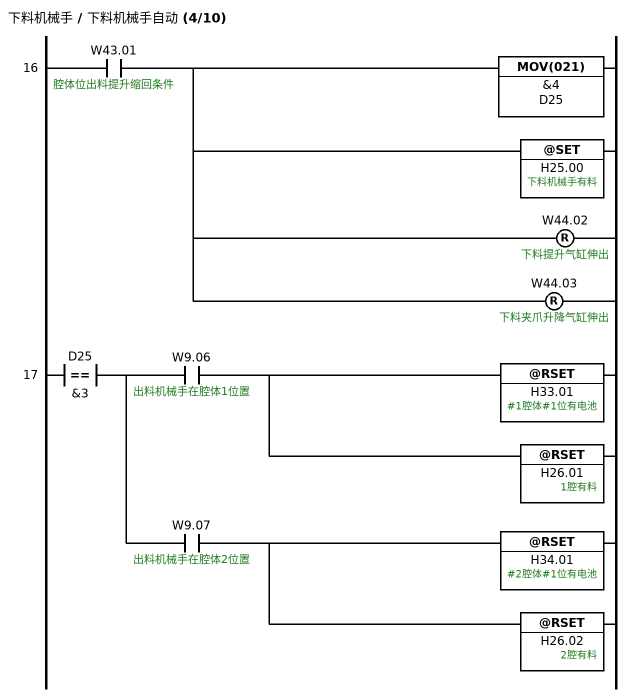
; [picture p168: 下料机械手 / 下料机械手自动, rungs 16-17]
; rung 16
LD W43.01  ; 腔体位出料提升缩回条件
MOV(021) &4 D25
@SET H25.00  ; 下料机械手有料
RSET W44.02  ; 下料提升气缸伸出
RSET W44.03  ; 下料夹爪升降气缸伸出
; rung 17
LD=(300) D25 &3
OUT TR0
AND W9.06  ; 出料机械手在腔体1位置
@RSET H33.01  ; #1腔体#1位有电池
@RSET H26.01  ; 1腔有料
LD TR0
AND W9.07  ; 出料机械手在腔体2位置
@RSET H34.01  ; #2腔体#1位有电池
@RSET H26.02  ; 2腔有料

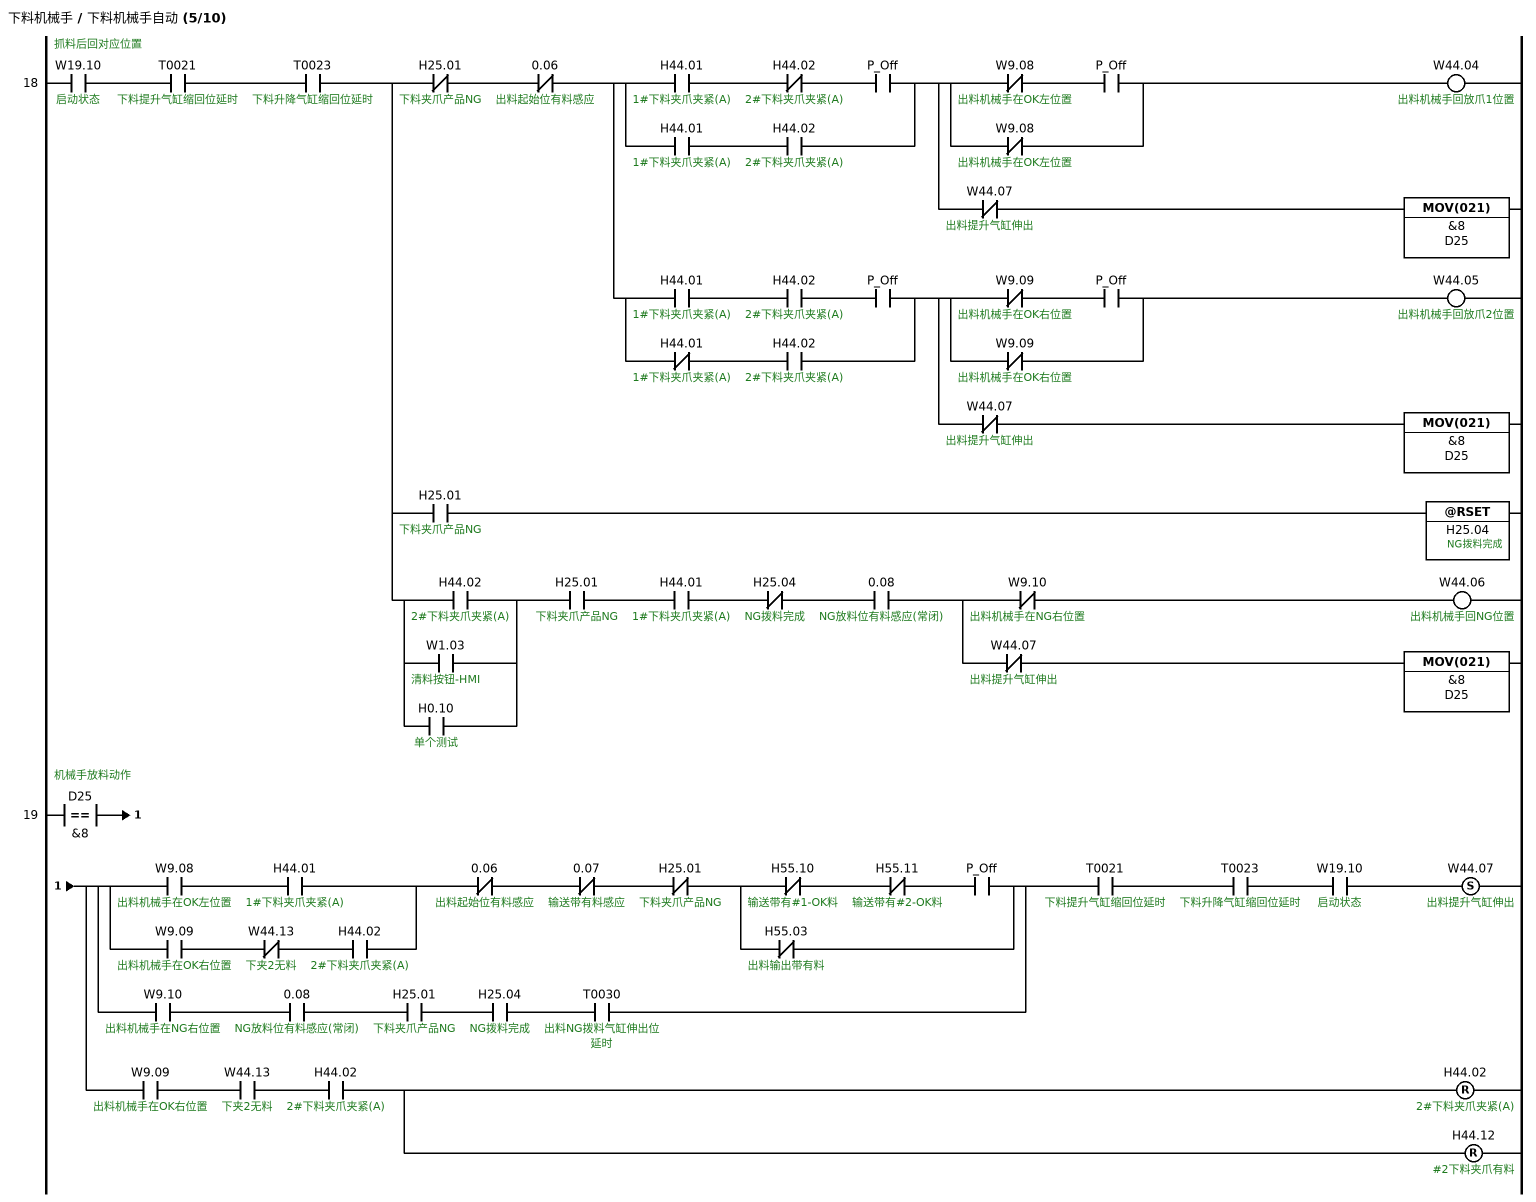
; rung 18: 抓料后回对应位置
LD W19.10  ; 启动状态
AND T0021  ; 下料提升气缸缩回位延时
AND T0023  ; 下料升降气缸缩回位延时
OUT TR0
ANDNOT H25.01  ; 下料夹爪产品NG
ANDNOT 0.06  ; 出料起始位有料感应
OUT TR1
LD H44.01  ; 1#下料夹爪夹紧(A)
ANDNOT H44.02  ; 2#下料夹爪夹紧(A)
AND P_Off
LD H44.01  ; 1#下料夹爪夹紧(A)
AND H44.02  ; 2#下料夹爪夹紧(A)
ORLD
ANDLD
OUT TR2
LDNOT W9.08  ; 出料机械手在OK左位置
AND P_Off
ORNOT W9.08  ; 出料机械手在OK左位置
ANDLD
OUT W44.04  ; 出料机械手回放爪1位置
LD TR2
ANDNOT W44.07  ; 出料提升气缸伸出
MOV(021) &8 D25
LD TR1
LD H44.01  ; 1#下料夹爪夹紧(A)
AND H44.02  ; 2#下料夹爪夹紧(A)
AND P_Off
LDNOT H44.01  ; 1#下料夹爪夹紧(A)
AND H44.02  ; 2#下料夹爪夹紧(A)
ORLD
ANDLD
OUT TR1
LDNOT W9.09  ; 出料机械手在OK右位置
AND P_Off
ORNOT W9.09  ; 出料机械手在OK右位置
ANDLD
OUT W44.05  ; 出料机械手回放爪2位置
LD TR1
ANDNOT W44.07  ; 出料提升气缸伸出
MOV(021) &8 D25
LD TR0
AND H25.01  ; 下料夹爪产品NG
@RSET H25.04  ; NG拨料完成
LD TR0
LD H44.02  ; 2#下料夹爪夹紧(A)
OR W1.03  ; 清料按钮-HMI
OR H0.10  ; 单个测试
ANDLD
AND H25.01  ; 下料夹爪产品NG
AND H44.01  ; 1#下料夹爪夹紧(A)
ANDNOT H25.04  ; NG拨料完成
AND 0.08  ; NG放料位有料感应(常闭)
OUT TR0
ANDNOT W9.10  ; 出料机械手在NG右位置
OUT W44.06  ; 出料机械手回NG位置
LD TR0
ANDNOT W44.07  ; 出料提升气缸伸出
MOV(021) &8 D25
; rung 19: 机械手放料动作
LD=(300) D25 &8
OUT TR0
LD W9.08  ; 出料机械手在OK左位置
AND H44.01  ; 1#下料夹爪夹紧(A)
LD W9.09  ; 出料机械手在OK右位置
ANDNOT W44.13  ; 下夹2无料
AND H44.02  ; 2#下料夹爪夹紧(A)
ORLD
ANDNOT 0.06  ; 出料起始位有料感应
ANDNOT 0.07  ; 输送带有料感应
ANDNOT H25.01  ; 下料夹爪产品NG
LDNOT H55.10  ; 输送带有#1-OK料
ANDNOT H55.11  ; 输送带有#2-OK料
AND P_Off
ORNOT H55.03  ; 出料输出带有料
ANDLD
LD W9.10  ; 出料机械手在NG右位置
AND 0.08  ; NG放料位有料感应(常闭)
AND H25.01  ; 下料夹爪产品NG
AND H25.04  ; NG拨料完成
AND T0030  ; 出料NG拨料气缸伸出位延时
ORLD
ANDLD
AND T0021  ; 下料提升气缸缩回位延时
AND T0023  ; 下料升降气缸缩回位延时
AND W19.10  ; 启动状态
SET W44.07  ; 出料提升气缸伸出
LD TR0
AND W9.09  ; 出料机械手在OK右位置
AND W44.13  ; 下夹2无料
AND H44.02  ; 2#下料夹爪夹紧(A)
RSET H44.02  ; 2#下料夹爪夹紧(A)
RSET H44.12  ; #2下料夹爪有料

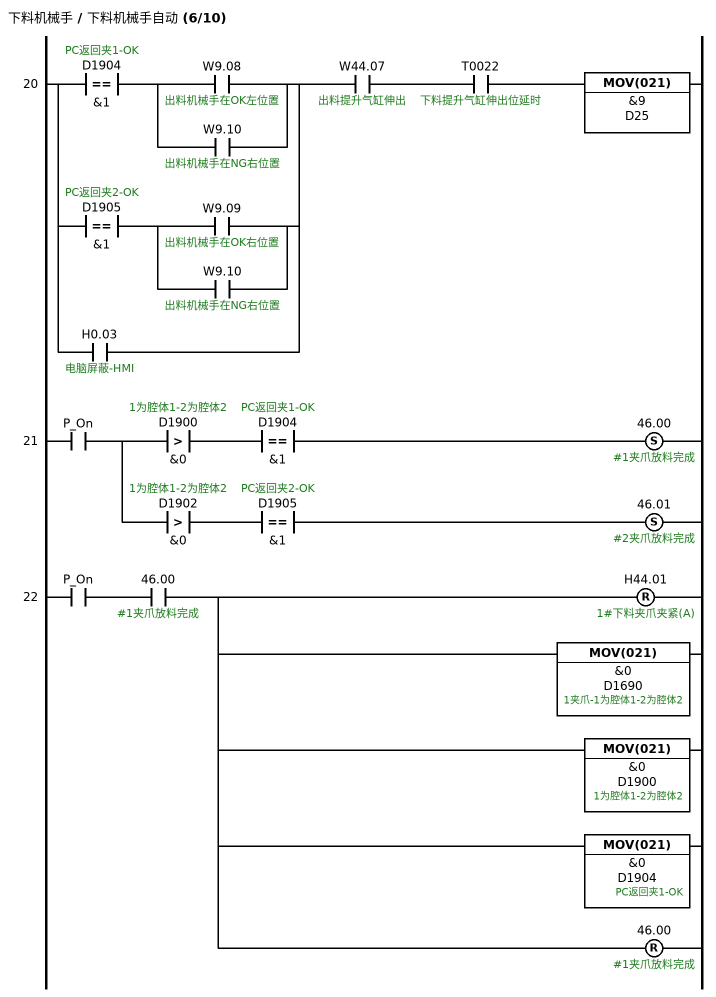
; rung 20
LD=(300) D1904 &1  ; PC返回夹1-OK
LD W9.08  ; 出料机械手在OK左位置
OR W9.10  ; 出料机械手在NG右位置
ANDLD
LD=(300) D1905 &1  ; PC返回夹2-OK
LD W9.09  ; 出料机械手在OK右位置
OR W9.10  ; 出料机械手在NG右位置
ANDLD
ORLD
OR H0.03  ; 电脑屏蔽-HMI
AND W44.07  ; 出料提升气缸伸出
AND T0022  ; 下料提升气缸伸出位延时
MOV(021) &9 D25
; rung 21
LD P_On
OUT TR0
AND>(320) D1900 &0  ; 1为腔体1-2为腔体2
AND=(300) D1904 &1  ; PC返回夹1-OK
SET 46.00  ; #1夹爪放料完成
LD TR0
AND>(320) D1902 &0  ; 1为腔体1-2为腔体2
AND=(300) D1905 &1  ; PC返回夹2-OK
SET 46.01  ; #2夹爪放料完成
; rung 22
LD P_On
AND 46.00  ; #1夹爪放料完成
RSET H44.01  ; 1#下料夹爪夹紧(A)
MOV(021) &0 D1690  ; 1夹爪-1为腔体1-2为腔体2
MOV(021) &0 D1900  ; 1为腔体1-2为腔体2
MOV(021) &0 D1904  ; PC返回夹1-OK
RSET 46.00  ; #1夹爪放料完成

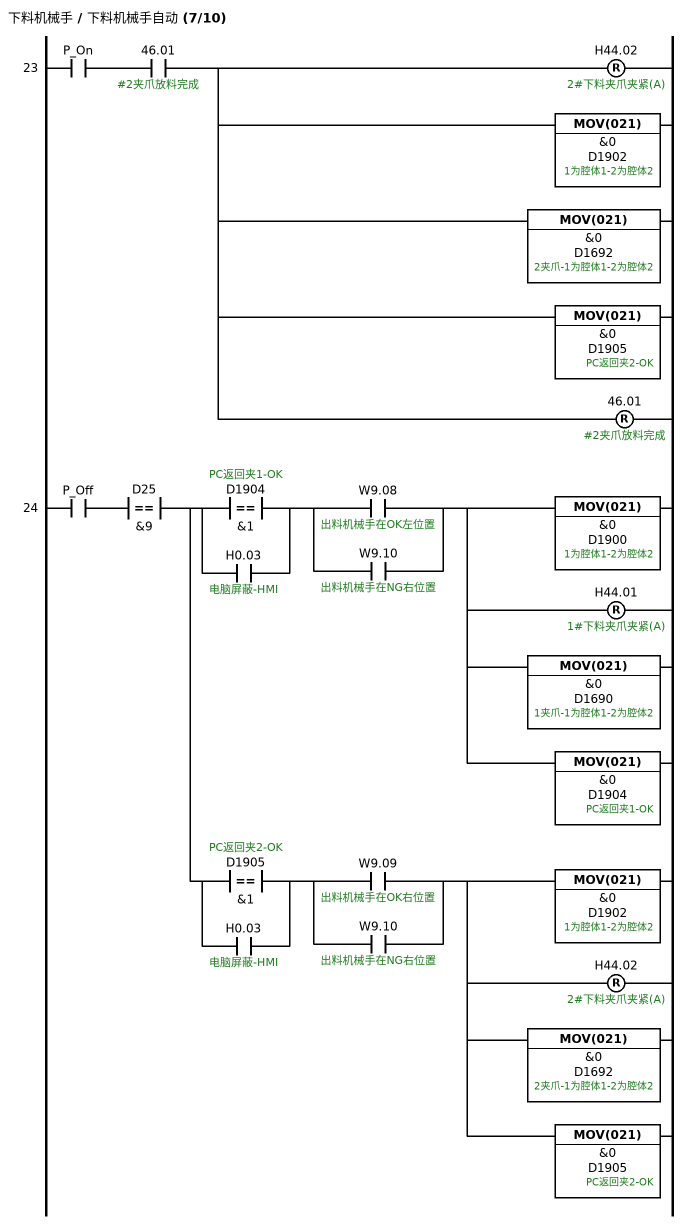
; rung 23
LD P_On
AND 46.01  ; #2夹爪放料完成
RSET H44.02  ; 2#下料夹爪夹紧(A)
MOV(021) &0 D1902  ; 1为腔体1-2为腔体2
MOV(021) &0 D1692  ; 2夹爪-1为腔体1-2为腔体2
MOV(021) &0 D1905  ; PC返回夹2-OK
RSET 46.01  ; #2夹爪放料完成
; rung 24
LD P_Off
AND=(300) D25 &9
OUT TR0
LD=(300) D1904 &1  ; PC返回夹1-OK
OR H0.03  ; 电脑屏蔽-HMI
ANDLD
LD W9.08  ; 出料机械手在OK左位置
OR W9.10  ; 出料机械手在NG右位置
ANDLD
MOV(021) &0 D1900  ; 1为腔体1-2为腔体2
RSET H44.01  ; 1#下料夹爪夹紧(A)
MOV(021) &0 D1690  ; 1夹爪-1为腔体1-2为腔体2
MOV(021) &0 D1904  ; PC返回夹1-OK
LD TR0
LD=(300) D1905 &1  ; PC返回夹2-OK
OR H0.03  ; 电脑屏蔽-HMI
ANDLD
LD W9.09  ; 出料机械手在OK右位置
OR W9.10  ; 出料机械手在NG右位置
ANDLD
MOV(021) &0 D1902  ; 1为腔体1-2为腔体2
RSET H44.02  ; 2#下料夹爪夹紧(A)
MOV(021) &0 D1692  ; 2夹爪-1为腔体1-2为腔体2
MOV(021) &0 D1905  ; PC返回夹2-OK

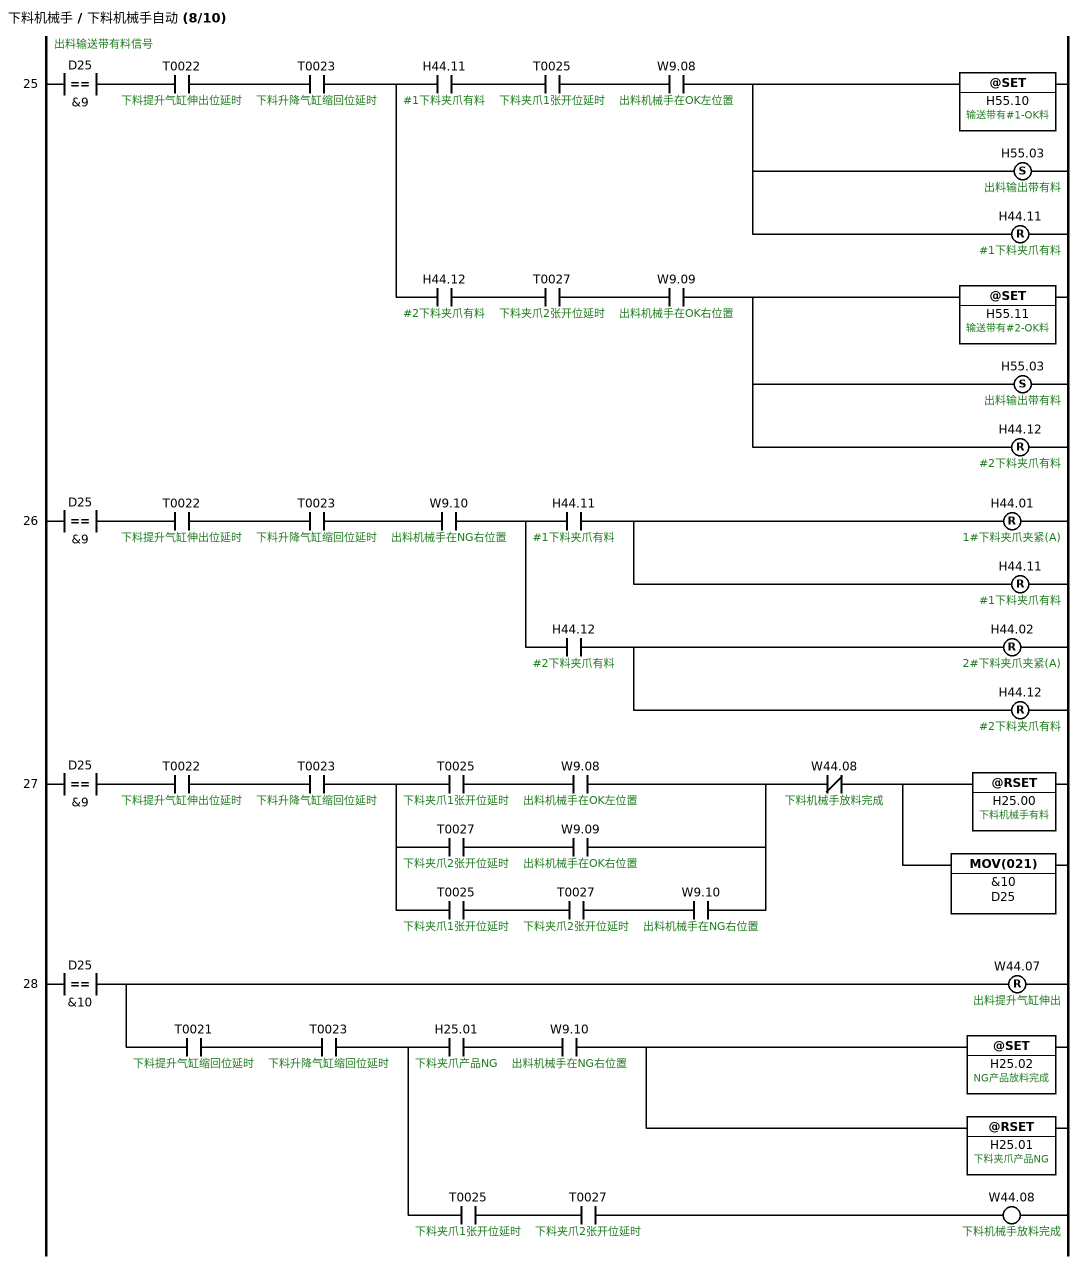
; rung 25: 出料输送带有料信号
LD=(300) D25 &9
AND T0022  ; 下料提升气缸伸出位延时
AND T0023  ; 下料升降气缸缩回位延时
OUT TR0
AND H44.11  ; #1下料夹爪有料
AND T0025  ; 下料夹爪1张开位延时
AND W9.08  ; 出料机械手在OK左位置
@SET H55.10  ; 输送带有#1-OK料
SET H55.03  ; 出料输出带有料
RSET H44.11  ; #1下料夹爪有料
LD TR0
AND H44.12  ; #2下料夹爪有料
AND T0027  ; 下料夹爪2张开位延时
AND W9.09  ; 出料机械手在OK右位置
@SET H55.11  ; 输送带有#2-OK料
SET H55.03  ; 出料输出带有料
RSET H44.12  ; #2下料夹爪有料
; rung 26
LD=(300) D25 &9
AND T0022  ; 下料提升气缸伸出位延时
AND T0023  ; 下料升降气缸缩回位延时
AND W9.10  ; 出料机械手在NG右位置
OUT TR0
AND H44.11  ; #1下料夹爪有料
RSET H44.01  ; 1#下料夹爪夹紧(A)
RSET H44.11  ; #1下料夹爪有料
LD TR0
AND H44.12  ; #2下料夹爪有料
RSET H44.02  ; 2#下料夹爪夹紧(A)
RSET H44.12  ; #2下料夹爪有料
; rung 27
LD=(300) D25 &9
AND T0022  ; 下料提升气缸伸出位延时
AND T0023  ; 下料升降气缸缩回位延时
LD T0025  ; 下料夹爪1张开位延时
AND W9.08  ; 出料机械手在OK左位置
LD T0027  ; 下料夹爪2张开位延时
AND W9.09  ; 出料机械手在OK右位置
ORLD
LD T0025  ; 下料夹爪1张开位延时
AND T0027  ; 下料夹爪2张开位延时
AND W9.10  ; 出料机械手在NG右位置
ORLD
ANDLD
ANDNOT W44.08  ; 下料机械手放料完成
@RSET H25.00  ; 下料机械手有料
MOV(021) &10 D25
; rung 28
LD=(300) D25 &10
RSET W44.07  ; 出料提升气缸伸出
AND T0021  ; 下料提升气缸缩回位延时
AND T0023  ; 下料升降气缸缩回位延时
OUT TR0
AND H25.01  ; 下料夹爪产品NG
AND W9.10  ; 出料机械手在NG右位置
@SET H25.02  ; NG产品放料完成
@RSET H25.01  ; 下料夹爪产品NG
LD TR0
AND T0025  ; 下料夹爪1张开位延时
AND T0027  ; 下料夹爪2张开位延时
OUT W44.08  ; 下料机械手放料完成

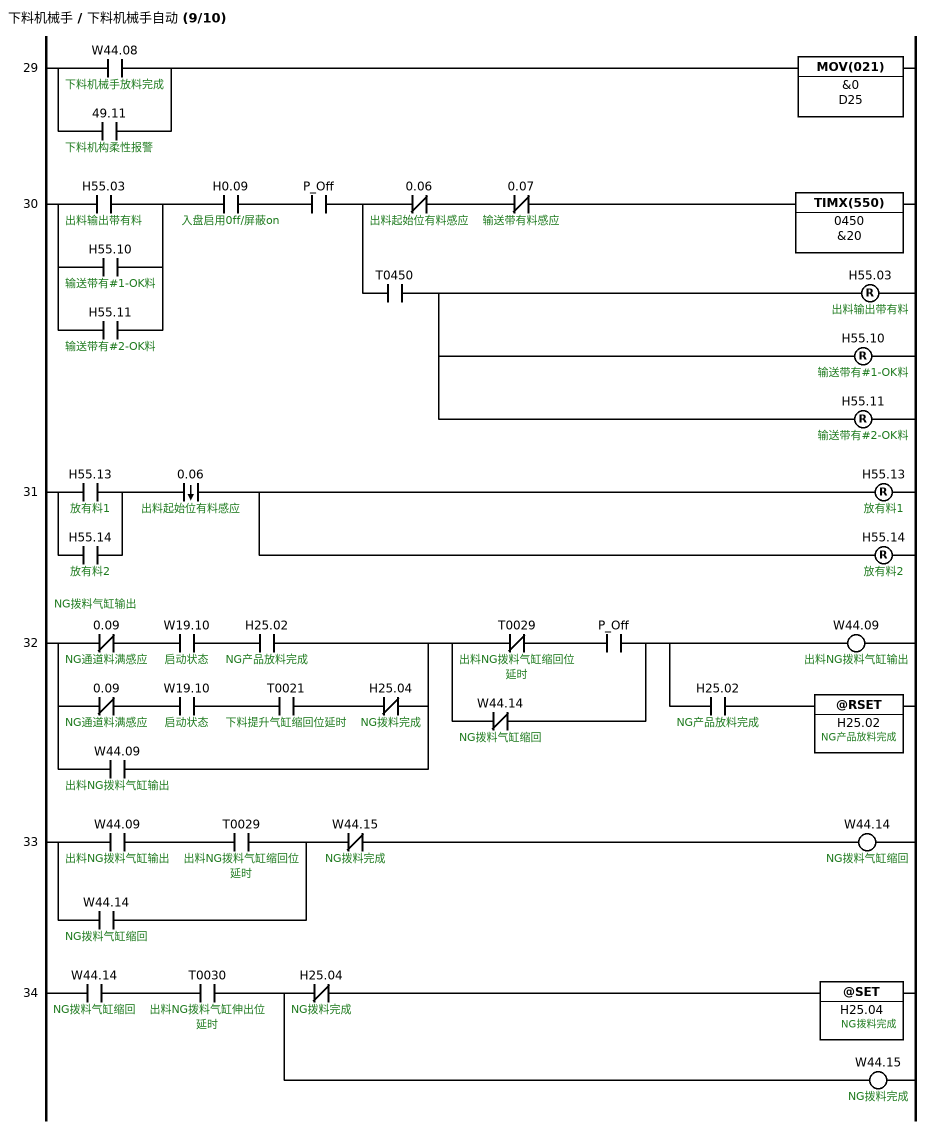
; rung 29
LD W44.08  ; 下料机械手放料完成
OR 49.11  ; 下料机构柔性报警
MOV(021) &0 D25
; rung 30
LD H55.03  ; 出料输出带有料
OR H55.10  ; 输送带有#1-OK料
OR H55.11  ; 输送带有#2-OK料
AND H0.09  ; 入盘启用0ff/屏蔽on
AND P_Off
OUT TR0
ANDNOT 0.06  ; 出料起始位有料感应
ANDNOT 0.07  ; 输送带有料感应
TIMX(550) 0450 &20
LD TR0
AND T0450
RSET H55.03  ; 出料输出带有料
RSET H55.10  ; 输送带有#1-OK料
RSET H55.11  ; 输送带有#2-OK料
; rung 31
LD H55.13  ; 放有料1
OR H55.14  ; 放有料2
%AND 0.06  ; 出料起始位有料感应
RSET H55.13  ; 放有料1
RSET H55.14  ; 放有料2
; rung 32: NG拨料气缸输出
LDNOT 0.09  ; NG通道料满感应
AND W19.10  ; 启动状态
AND H25.02  ; NG产品放料完成
LDNOT 0.09  ; NG通道料满感应
AND W19.10  ; 启动状态
AND T0021  ; 下料提升气缸缩回位延时
ANDNOT H25.04  ; NG拨料完成
ORLD
OR W44.09  ; 出料NG拨料气缸输出
LDNOT T0029  ; 出料NG拨料气缸缩回位延时
AND P_Off
ORNOT W44.14  ; NG拨料气缸缩回
ANDLD
OUT W44.09  ; 出料NG拨料气缸输出
AND H25.02  ; NG产品放料完成
@RSET H25.02  ; NG产品放料完成
; rung 33
LD W44.09  ; 出料NG拨料气缸输出
AND T0029  ; 出料NG拨料气缸缩回位延时
OR W44.14  ; NG拨料气缸缩回
ANDNOT W44.15  ; NG拨料完成
OUT W44.14  ; NG拨料气缸缩回
; rung 34
LD W44.14  ; NG拨料气缸缩回
AND T0030  ; 出料NG拨料气缸伸出位延时
OUT TR0
ANDNOT H25.04  ; NG拨料完成
@SET H25.04  ; NG拨料完成
LD TR0
OUT W44.15  ; NG拨料完成

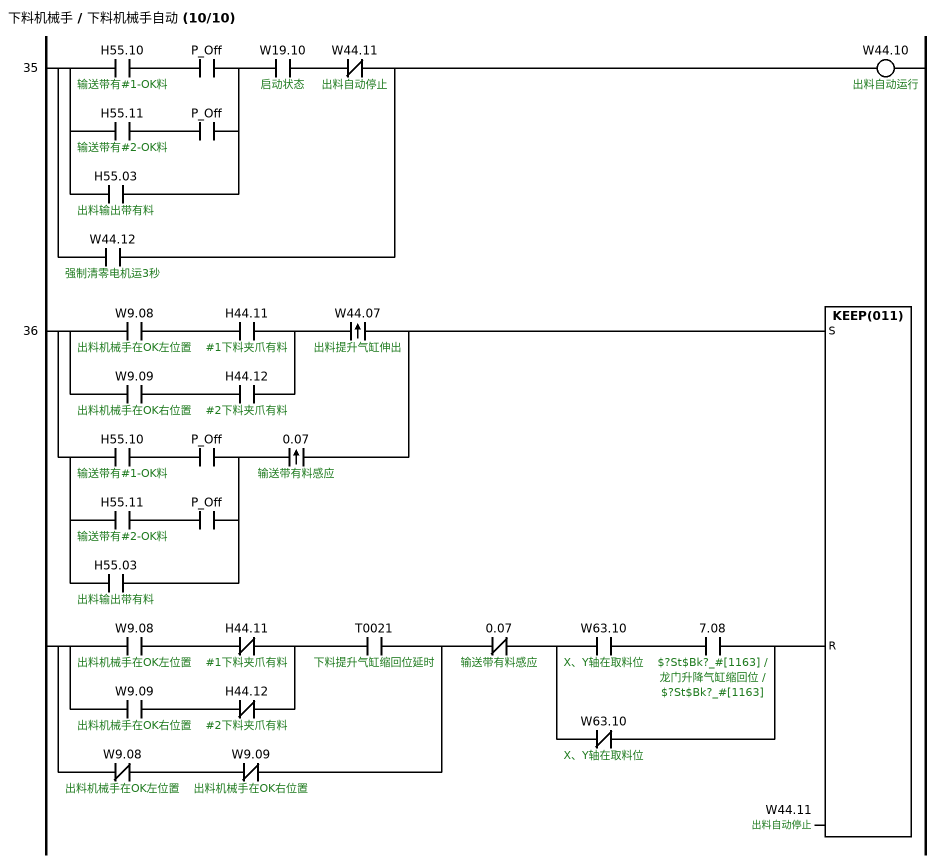
; rung 35
LD H55.10  ; 输送带有#1-OK料
AND P_Off
LD H55.11  ; 输送带有#2-OK料
AND P_Off
ORLD
OR H55.03  ; 出料输出带有料
AND W19.10  ; 启动状态
ANDNOT W44.11  ; 出料自动停止
OR W44.12  ; 强制清零电机运3秒
OUT W44.10  ; 出料自动运行
; rung 36
LD W9.08  ; 出料机械手在OK左位置
AND H44.11  ; #1下料夹爪有料
LD W9.09  ; 出料机械手在OK右位置
AND H44.12  ; #2下料夹爪有料
ORLD
@AND W44.07  ; 出料提升气缸伸出
LD H55.10  ; 输送带有#1-OK料
AND P_Off
LD H55.11  ; 输送带有#2-OK料
AND P_Off
ORLD
OR H55.03  ; 出料输出带有料
@AND 0.07  ; 输送带有料感应
ORLD
LD W9.08  ; 出料机械手在OK左位置
ANDNOT H44.11  ; #1下料夹爪有料
LD W9.09  ; 出料机械手在OK右位置
ANDNOT H44.12  ; #2下料夹爪有料
ORLD
AND T0021  ; 下料提升气缸缩回位延时
LDNOT W9.08  ; 出料机械手在OK左位置
ANDNOT W9.09  ; 出料机械手在OK右位置
ORLD
ANDNOT 0.07  ; 输送带有料感应
LD W63.10  ; X、Y轴在取料位
AND 7.08  ; $?St$Bk?_#[1163] / 龙门升降气缸缩回位 / $?St$Bk?_#[1163]
ORNOT W63.10  ; X、Y轴在取料位
ANDLD
KEEP(011) W44.11  ; 出料自动停止

### Section 伺服参数

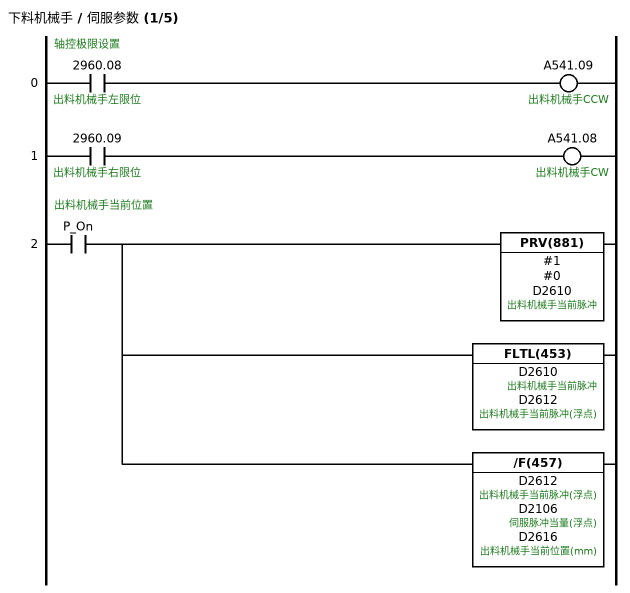
; rung 0: 轴控极限设置
LD 2960.08  ; 出料机械手左限位
OUT A541.09  ; 出料机械手CCW
; rung 1
LD 2960.09  ; 出料机械手右限位
OUT A541.08  ; 出料机械手CW
; rung 2: 出料机械手当前位置
LD P_On
PRV(881) #1 #0 D2610  ; 出料机械手当前脉冲
FLTL(453) D2610 D2612  ; 出料机械手当前脉冲, 出料机械手当前脉冲(浮点)
/F(457) D2612 D2106 D2616  ; 出料机械手当前脉冲(浮点), 伺服脉冲当量(浮点), 出料机械手当前位置(mm)

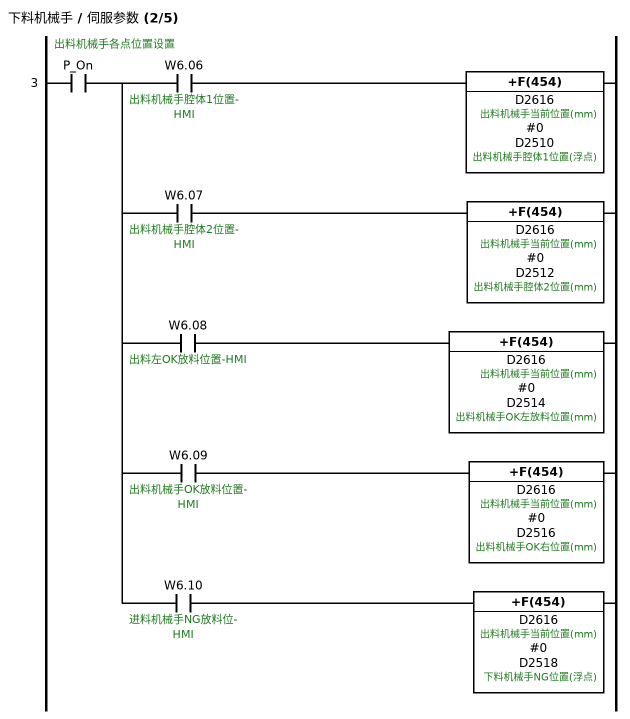
; rung 3: 出料机械手各点位置设置
LD P_On
OUT TR0
AND W6.06  ; 出料机械手腔体1位置-HMI
+F(454) D2616 #0 D2510  ; 出料机械手当前位置(mm), 出料机械手腔体1位置(浮点)
LD TR0
AND W6.07  ; 出料机械手腔体2位置-HMI
+F(454) D2616 #0 D2512  ; 出料机械手当前位置(mm), 出料机械手腔体2位置(mm)
LD TR0
AND W6.08  ; 出料左OK放料位置-HMI
+F(454) D2616 #0 D2514  ; 出料机械手当前位置(mm), 出料机械手OK左放料位置(mm)
LD TR0
AND W6.09  ; 出料机械手OK放料位置-HMI
+F(454) D2616 #0 D2516  ; 出料机械手当前位置(mm), 出料机械手OK右位置(mm)
LD TR0
AND W6.10  ; 进料机械手NG放料位-HMI
+F(454) D2616 #0 D2518  ; 出料机械手当前位置(mm), 下料机械手NG位置(浮点)

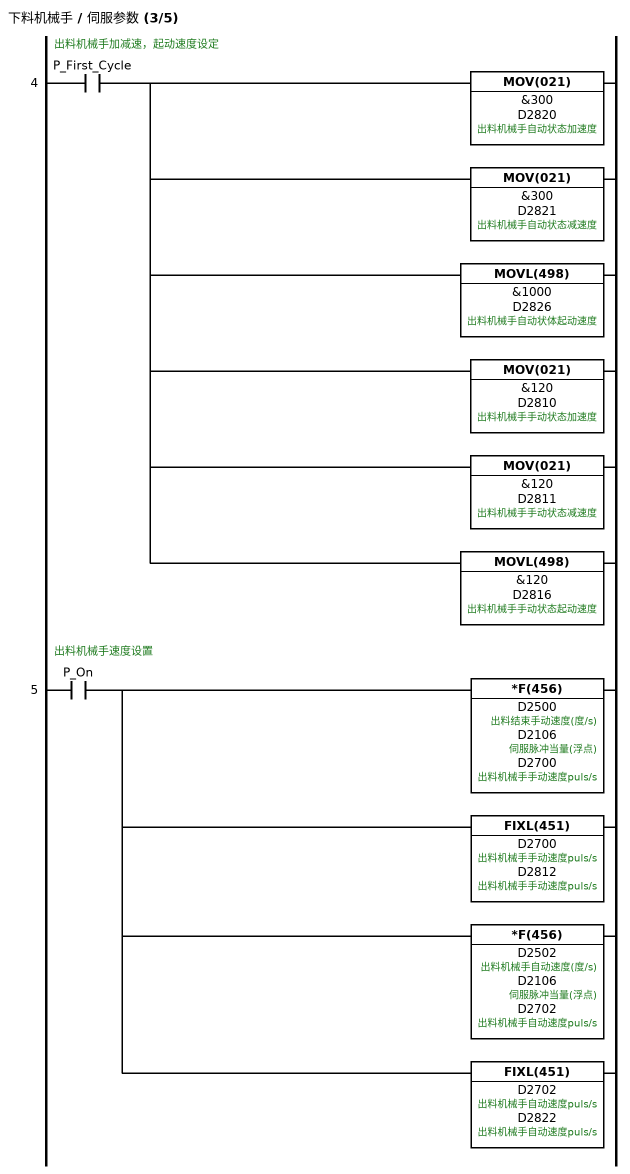
; rung 4: 出料机械手加减速，起动速度设定
LD P_First_Cycle
MOV(021) &300 D2820  ; 出料机械手自动状态加速度
MOV(021) &300 D2821  ; 出料机械手自动状态减速度
MOVL(498) &1000 D2826  ; 出料机械手自动状体起动速度
MOV(021) &120 D2810  ; 出料机械手手动状态加速度
MOV(021) &120 D2811  ; 出料机械手手动状态减速度
MOVL(498) &120 D2816  ; 出料机械手手动状态起动速度
; rung 5: 出料机械手速度设置
LD P_On
*F(456) D2500 D2106 D2700  ; 出料结束手动速度(度/s), 伺服脉冲当量(浮点), 出料机械手手动速度puls/s
FIXL(451) D2700 D2812  ; 出料机械手手动速度puls/s
*F(456) D2502 D2106 D2702  ; 出料机械手自动速度(度/s), 伺服脉冲当量(浮点), 出料机械手自动速度puls/s
FIXL(451) D2702 D2822  ; 出料机械手自动速度puls/s

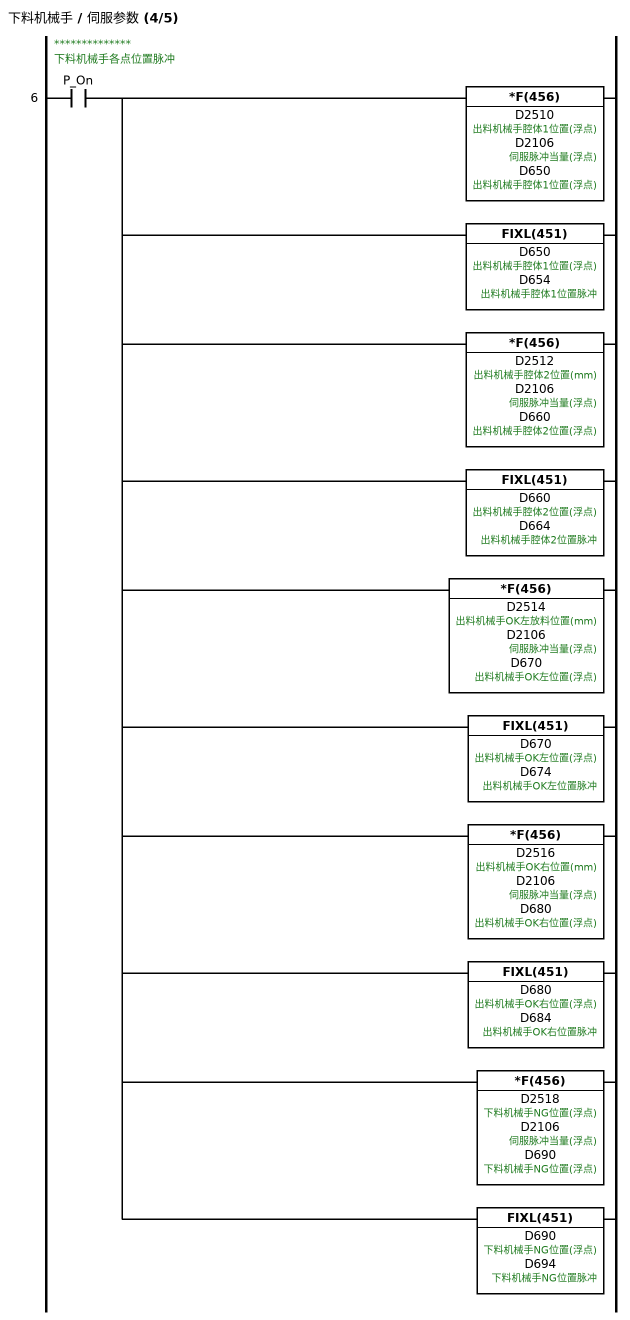
; rung 6: ************** / 下料机械手各点位置脉冲
LD P_On
*F(456) D2510 D2106 D650  ; 出料机械手腔体1位置(浮点), 伺服脉冲当量(浮点)
FIXL(451) D650 D654  ; 出料机械手腔体1位置(浮点), 出料机械手腔体1位置脉冲
*F(456) D2512 D2106 D660  ; 出料机械手腔体2位置(mm), 伺服脉冲当量(浮点), 出料机械手腔体2位置(浮点)
FIXL(451) D660 D664  ; 出料机械手腔体2位置(浮点), 出料机械手腔体2位置脉冲
*F(456) D2514 D2106 D670  ; 出料机械手OK左放料位置(mm), 伺服脉冲当量(浮点), 出料机械手OK左位置(浮点)
FIXL(451) D670 D674  ; 出料机械手OK左位置(浮点), 出料机械手OK左位置脉冲
*F(456) D2516 D2106 D680  ; 出料机械手OK右位置(mm), 伺服脉冲当量(浮点), 出料机械手OK右位置(浮点)
FIXL(451) D680 D684  ; 出料机械手OK右位置(浮点), 出料机械手OK右位置脉冲
*F(456) D2518 D2106 D690  ; 下料机械手NG位置(浮点), 伺服脉冲当量(浮点)
FIXL(451) D690 D694  ; 下料机械手NG位置(浮点), 下料机械手NG位置脉冲

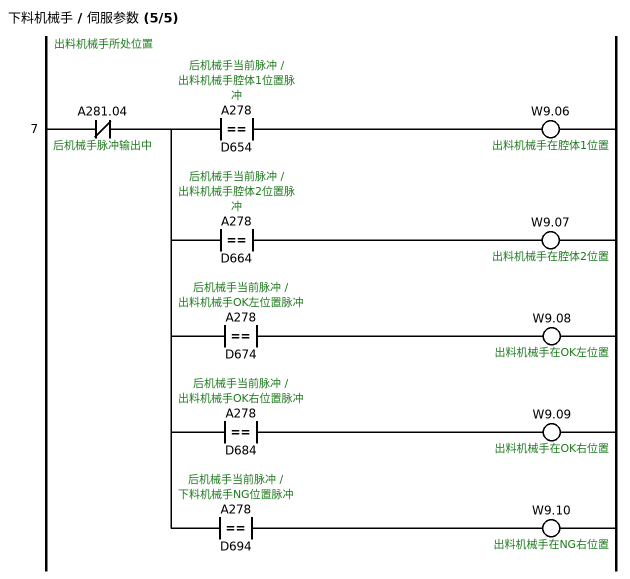
; rung 7: 出料机械手所处位置
LDNOT A281.04  ; 后机械手脉冲输出中
OUT TR0
AND=SL(303) A278 D654  ; 后机械手当前脉冲, 出料机械手腔体1位置脉冲
OUT W9.06  ; 出料机械手在腔体1位置
LD TR0
AND=SL(303) A278 D664  ; 后机械手当前脉冲, 出料机械手腔体2位置脉冲
OUT W9.07  ; 出料机械手在腔体2位置
LD TR0
AND=SL(303) A278 D674  ; 后机械手当前脉冲, 出料机械手OK左位置脉冲
OUT W9.08  ; 出料机械手在OK左位置
LD TR0
AND=SL(303) A278 D684  ; 后机械手当前脉冲, 出料机械手OK右位置脉冲
OUT W9.09  ; 出料机械手在OK右位置
LD TR0
AND=SL(303) A278 D694  ; 后机械手当前脉冲, 下料机械手NG位置脉冲
OUT W9.10  ; 出料机械手在NG右位置

### Section 外部输出及轴控运动

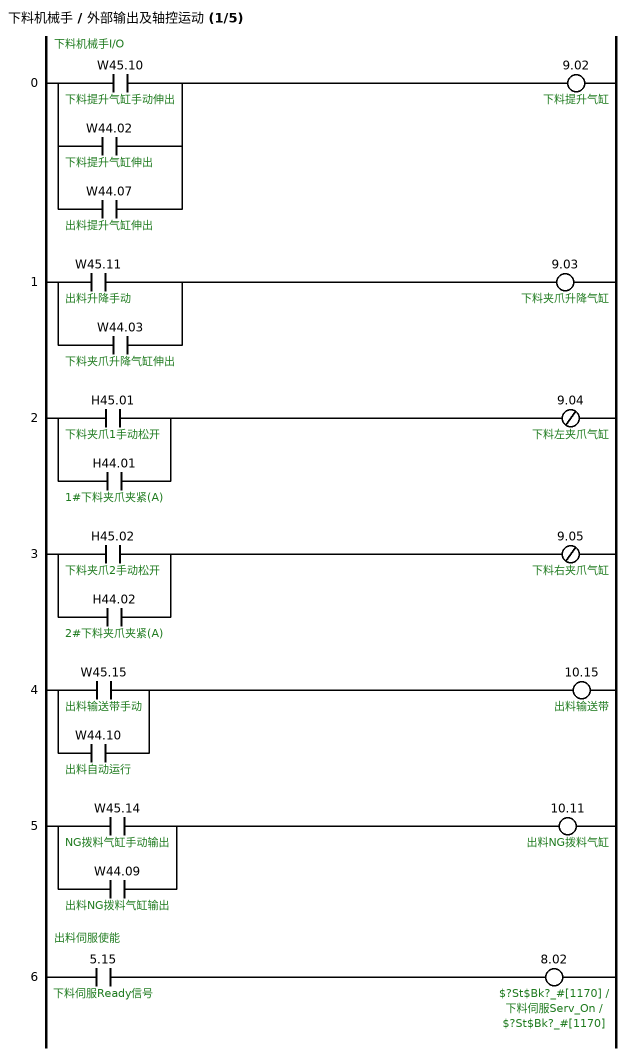
; rung 0: 下料机械手I/O
LD W45.10  ; 下料提升气缸手动伸出
OR W44.02  ; 下料提升气缸伸出
OR W44.07  ; 出料提升气缸伸出
OUT 9.02  ; 下料提升气缸
; rung 1
LD W45.11  ; 出料升降手动
OR W44.03  ; 下料夹爪升降气缸伸出
OUT 9.03  ; 下料夹爪升降气缸
; rung 2
LD H45.01  ; 下料夹爪1手动松开
OR H44.01  ; 1#下料夹爪夹紧(A)
OUTNOT 9.04  ; 下料左夹爪气缸
; rung 3
LD H45.02  ; 下料夹爪2手动松开
OR H44.02  ; 2#下料夹爪夹紧(A)
OUTNOT 9.05  ; 下料右夹爪气缸
; rung 4
LD W45.15  ; 出料输送带手动
OR W44.10  ; 出料自动运行
OUT 10.15  ; 出料输送带
; rung 5
LD W45.14  ; NG拨料气缸手动输出
OR W44.09  ; 出料NG拨料气缸输出
OUT 10.11  ; 出料NG拨料气缸
; rung 6: 出料伺服使能
LD 5.15  ; 下料伺服Ready信号
OUT 8.02  ; $?St$Bk?_#[1170] / 下料伺服Serv_On / $?St$Bk?_#[1170]

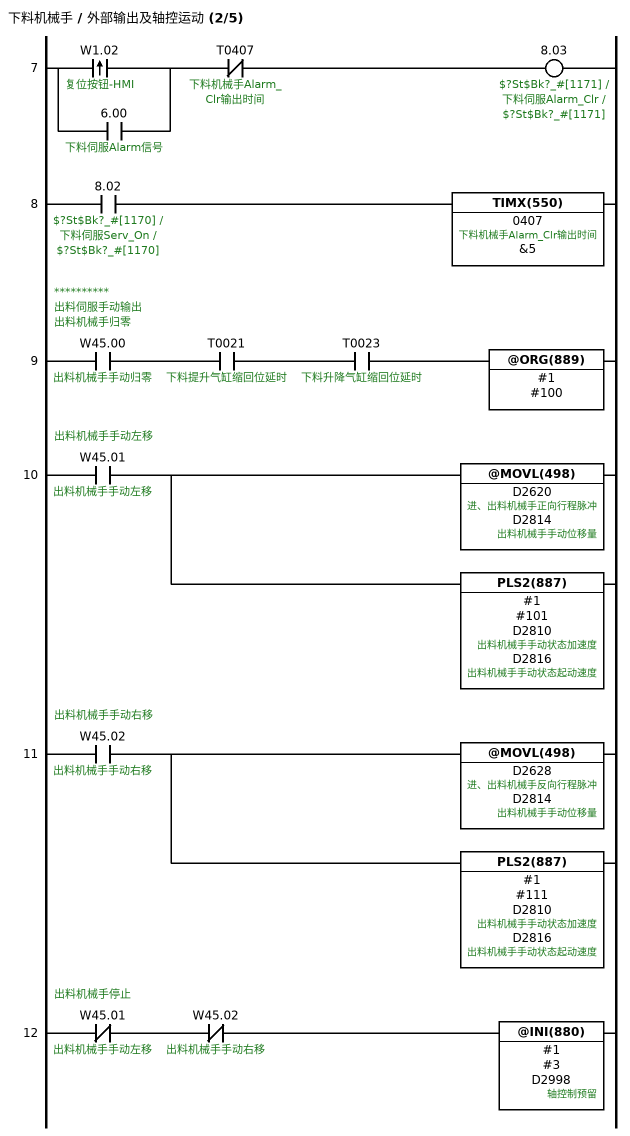
; rung 7
@LD W1.02  ; 复位按钮-HMI
OR 6.00  ; 下料伺服Alarm信号
ANDNOT T0407  ; 下料机械手Alarm_Clr输出时间
OUT 8.03  ; $?St$Bk?_#[1171] / 下料伺服Alarm_Clr / $?St$Bk?_#[1171]
; rung 8
LD 8.02  ; $?St$Bk?_#[1170] / 下料伺服Serv_On / $?St$Bk?_#[1170]
TIMX(550) 0407 &5  ; 下料机械手Alarm_Clr输出时间
; rung 9: ********** / 出料伺服手动输出 / 出料机械手归零
LD W45.00  ; 出料机械手手动归零
AND T0021  ; 下料提升气缸缩回位延时
AND T0023  ; 下料升降气缸缩回位延时
@ORG(889) #1 #100
; rung 10: 出料机械手手动左移
LD W45.01  ; 出料机械手手动左移
@MOVL(498) D2620 D2814  ; 进、出料机械手正向行程脉冲, 出料机械手手动位移量
PLS2(887) #1 #101 D2810 D2816  ; 出料机械手手动状态加速度, 出料机械手手动状态起动速度
; rung 11: 出料机械手手动右移
LD W45.02  ; 出料机械手手动右移
@MOVL(498) D2628 D2814  ; 进、出料机械手反向行程脉冲, 出料机械手手动位移量
PLS2(887) #1 #111 D2810 D2816  ; 出料机械手手动状态加速度, 出料机械手手动状态起动速度
; rung 12: 出料机械手停止
LDNOT W45.01  ; 出料机械手手动左移
ANDNOT W45.02  ; 出料机械手手动右移
@INI(880) #1 #3 D2998  ; 轴控制预留

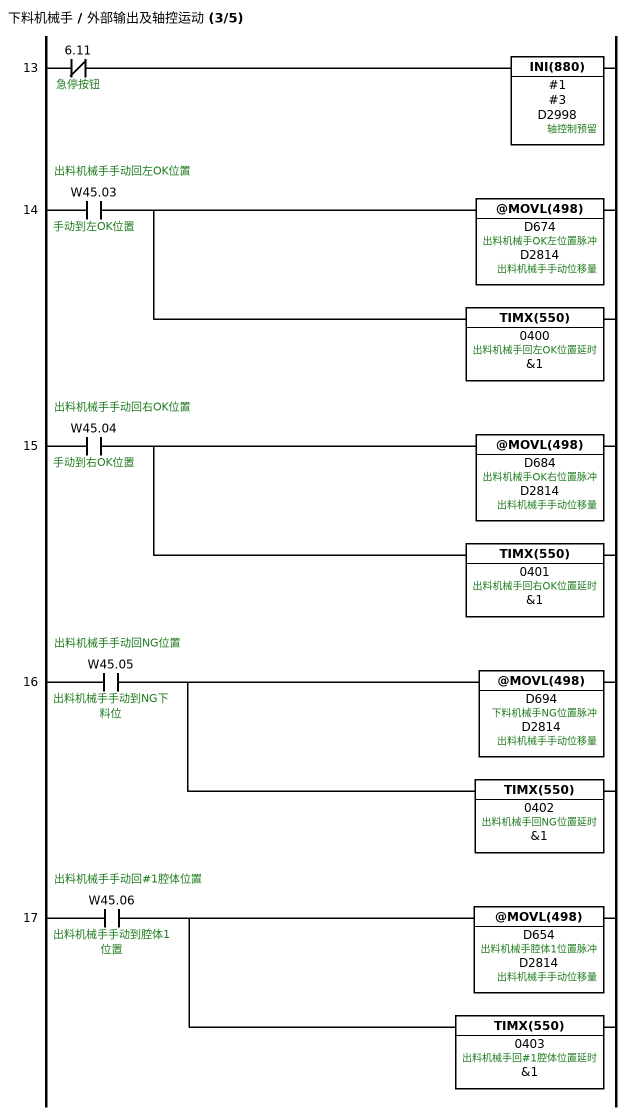
; rung 13
LDNOT 6.11  ; 急停按钮
INI(880) #1 #3 D2998  ; 轴控制预留
; rung 14: 出料机械手手动回左OK位置
LD W45.03  ; 手动到左OK位置
@MOVL(498) D674 D2814  ; 出料机械手OK左位置脉冲, 出料机械手手动位移量
TIMX(550) 0400 &1  ; 出料机械手回左OK位置延时
; rung 15: 出料机械手手动回右OK位置
LD W45.04  ; 手动到右OK位置
@MOVL(498) D684 D2814  ; 出料机械手OK右位置脉冲, 出料机械手手动位移量
TIMX(550) 0401 &1  ; 出料机械手回右OK位置延时
; rung 16: 出料机械手手动回NG位置
LD W45.05  ; 出料机械手手动到NG下料位
@MOVL(498) D694 D2814  ; 下料机械手NG位置脉冲, 出料机械手手动位移量
TIMX(550) 0402 &1  ; 出料机械手回NG位置延时
; rung 17: 出料机械手手动回#1腔体位置
LD W45.06  ; 出料机械手手动到腔体1位置
@MOVL(498) D654 D2814  ; 出料机械手腔体1位置脉冲, 出料机械手手动位移量
TIMX(550) 0403 &1  ; 出料机械手回#1腔体位置延时

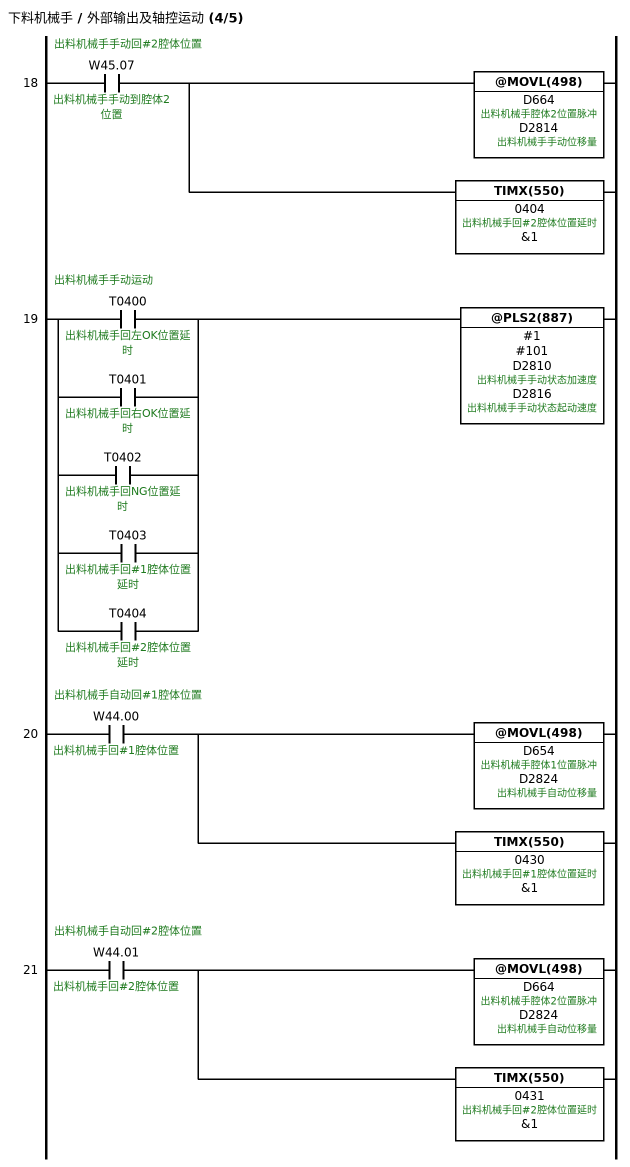
; rung 18: 出料机械手手动回#2腔体位置
LD W45.07  ; 出料机械手手动到腔体2位置
@MOVL(498) D664 D2814  ; 出料机械手腔体2位置脉冲, 出料机械手手动位移量
TIMX(550) 0404 &1  ; 出料机械手回#2腔体位置延时
; rung 19: 出料机械手手动运动
LD T0400  ; 出料机械手回左OK位置延时
OR T0401  ; 出料机械手回右OK位置延时
OR T0402  ; 出料机械手回NG位置延时
OR T0403  ; 出料机械手回#1腔体位置延时
OR T0404  ; 出料机械手回#2腔体位置延时
@PLS2(887) #1 #101 D2810 D2816  ; 出料机械手手动状态加速度, 出料机械手手动状态起动速度
; rung 20: 出料机械手自动回#1腔体位置
LD W44.00  ; 出料机械手回#1腔体位置
@MOVL(498) D654 D2824  ; 出料机械手腔体1位置脉冲, 出料机械手自动位移量
TIMX(550) 0430 &1  ; 出料机械手回#1腔体位置延时
; rung 21: 出料机械手自动回#2腔体位置
LD W44.01  ; 出料机械手回#2腔体位置
@MOVL(498) D664 D2824  ; 出料机械手腔体2位置脉冲, 出料机械手自动位移量
TIMX(550) 0431 &1  ; 出料机械手回#2腔体位置延时

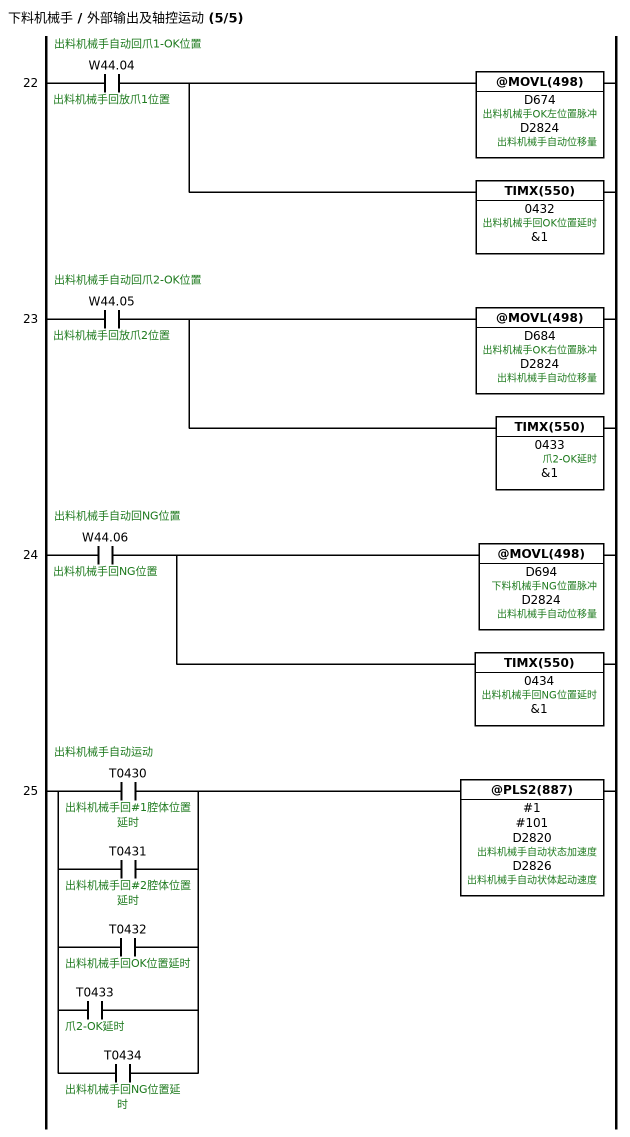
; rung 22: 出料机械手自动回爪1-OK位置
LD W44.04  ; 出料机械手回放爪1位置
@MOVL(498) D674 D2824  ; 出料机械手OK左位置脉冲, 出料机械手自动位移量
TIMX(550) 0432 &1  ; 出料机械手回OK位置延时
; rung 23: 出料机械手自动回爪2-OK位置
LD W44.05  ; 出料机械手回放爪2位置
@MOVL(498) D684 D2824  ; 出料机械手OK右位置脉冲, 出料机械手自动位移量
TIMX(550) 0433 &1  ; 爪2-OK延时
; rung 24: 出料机械手自动回NG位置
LD W44.06  ; 出料机械手回NG位置
@MOVL(498) D694 D2824  ; 下料机械手NG位置脉冲, 出料机械手自动位移量
TIMX(550) 0434 &1  ; 出料机械手回NG位置延时
; rung 25: 出料机械手自动运动
LD T0430  ; 出料机械手回#1腔体位置延时
OR T0431  ; 出料机械手回#2腔体位置延时
OR T0432  ; 出料机械手回OK位置延时
OR T0433  ; 爪2-OK延时
OR T0434  ; 出料机械手回NG位置延时
@PLS2(887) #1 #101 D2820 D2826  ; 出料机械手自动状态加速度, 出料机械手自动状体起动速度

### Section 自动报警

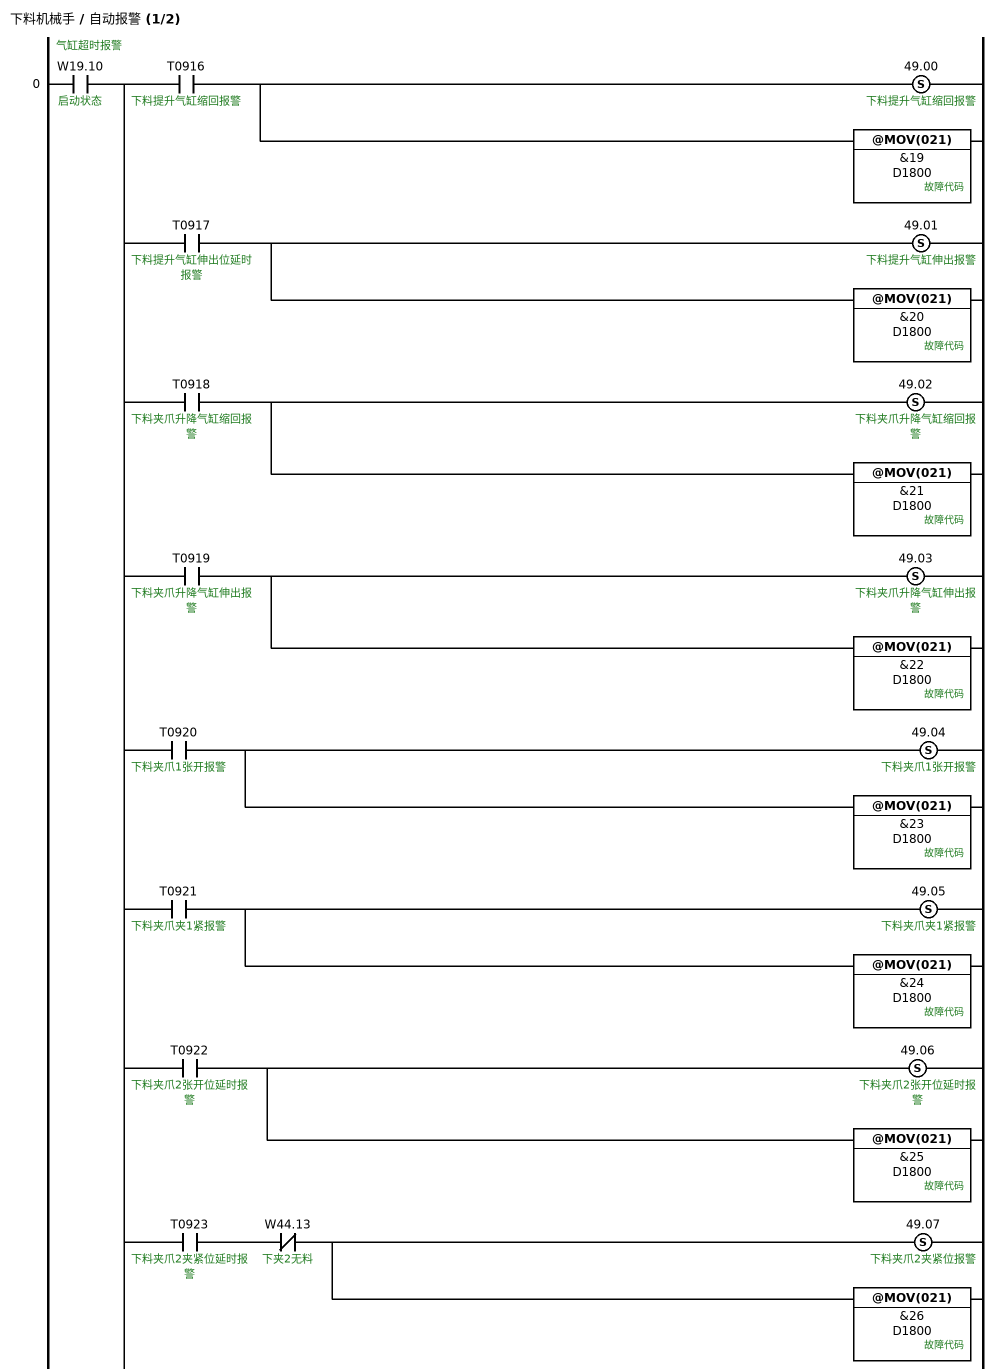

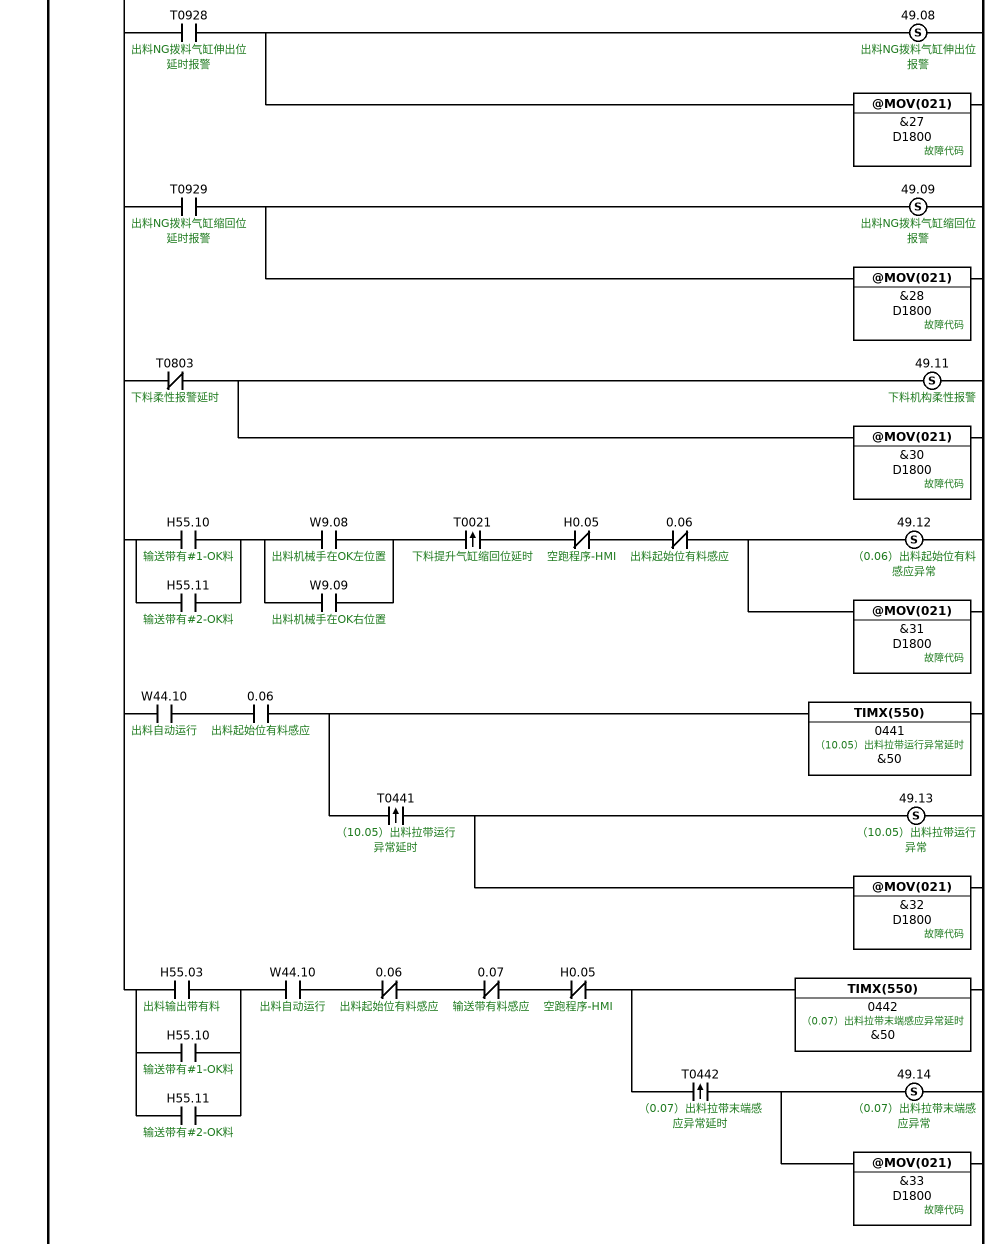
; rung 0: 气缸超时报警
LD W19.10  ; 启动状态
OUT TR0
AND T0916  ; 下料提升气缸缩回报警
SET 49.00  ; 下料提升气缸缩回报警
@MOV(021) &19 D1800  ; 故障代码
LD TR0
AND T0917  ; 下料提升气缸伸出位延时报警
SET 49.01  ; 下料提升气缸伸出报警
@MOV(021) &20 D1800  ; 故障代码
LD TR0
AND T0918  ; 下料夹爪升降气缸缩回报警
SET 49.02  ; 下料夹爪升降气缸缩回报警
@MOV(021) &21 D1800  ; 故障代码
LD TR0
AND T0919  ; 下料夹爪升降气缸伸出报警
SET 49.03  ; 下料夹爪升降气缸伸出报警
@MOV(021) &22 D1800  ; 故障代码
LD TR0
AND T0920  ; 下料夹爪1张开报警
SET 49.04  ; 下料夹爪1张开报警
@MOV(021) &23 D1800  ; 故障代码
LD TR0
AND T0921  ; 下料夹爪夹1紧报警
SET 49.05  ; 下料夹爪夹1紧报警
@MOV(021) &24 D1800  ; 故障代码
LD TR0
AND T0922  ; 下料夹爪2张开位延时报警
SET 49.06  ; 下料夹爪2张开位延时报警
@MOV(021) &25 D1800  ; 故障代码
LD TR0
AND T0923  ; 下料夹爪2夹紧位延时报警
ANDNOT W44.13  ; 下夹2无料
SET 49.07  ; 下料夹爪2夹紧位报警
@MOV(021) &26 D1800  ; 故障代码
LD TR0
AND T0928  ; 出料NG拨料气缸伸出位延时报警
SET 49.08  ; 出料NG拨料气缸伸出位报警
@MOV(021) &27 D1800  ; 故障代码
LD TR0
AND T0929  ; 出料NG拨料气缸缩回位延时报警
SET 49.09  ; 出料NG拨料气缸缩回位报警
@MOV(021) &28 D1800  ; 故障代码
LD TR0
ANDNOT T0803  ; 下料柔性报警延时
SET 49.11  ; 下料机构柔性报警
@MOV(021) &30 D1800  ; 故障代码
LD TR0
LD H55.10  ; 输送带有#1-OK料
OR H55.11  ; 输送带有#2-OK料
ANDLD
LD W9.08  ; 出料机械手在OK左位置
OR W9.09  ; 出料机械手在OK右位置
ANDLD
@AND T0021  ; 下料提升气缸缩回位延时
ANDNOT H0.05  ; 空跑程序-HMI
ANDNOT 0.06  ; 出料起始位有料感应
SET 49.12  ; （0.06）出料起始位有料感应异常
@MOV(021) &31 D1800  ; 故障代码
LD TR0
AND W44.10  ; 出料自动运行
AND 0.06  ; 出料起始位有料感应
TIMX(550) 0441 &50  ; （10.05）出料拉带运行异常延时
@AND T0441  ; （10.05）出料拉带运行异常延时
SET 49.13  ; （10.05）出料拉带运行异常
@MOV(021) &32 D1800  ; 故障代码
LD TR0
LD H55.03  ; 出料输出带有料
OR H55.10  ; 输送带有#1-OK料
OR H55.11  ; 输送带有#2-OK料
ANDLD
AND W44.10  ; 出料自动运行
ANDNOT 0.06  ; 出料起始位有料感应
ANDNOT 0.07  ; 输送带有料感应
ANDNOT H0.05  ; 空跑程序-HMI
TIMX(550) 0442 &50  ; （0.07）出料拉带末端感应异常延时
@AND T0442  ; （0.07）出料拉带末端感应异常延时
SET 49.14  ; （0.07）出料拉带末端感应异常
@MOV(021) &33 D1800  ; 故障代码

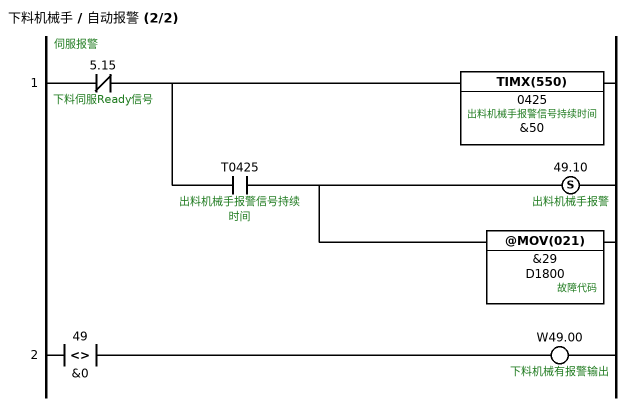
; rung 1: 伺服报警
LDNOT 5.15  ; 下料伺服Ready信号
TIMX(550) 0425 &50  ; 出料机械手报警信号持续时间
AND T0425  ; 出料机械手报警信号持续时间
SET 49.10  ; 出料机械手报警
@MOV(021) &29 D1800  ; 故障代码
; rung 2
LD<>(305) 49 &0
OUT W49.00  ; 下料机械有报警输出

### Section 下料机械手复位

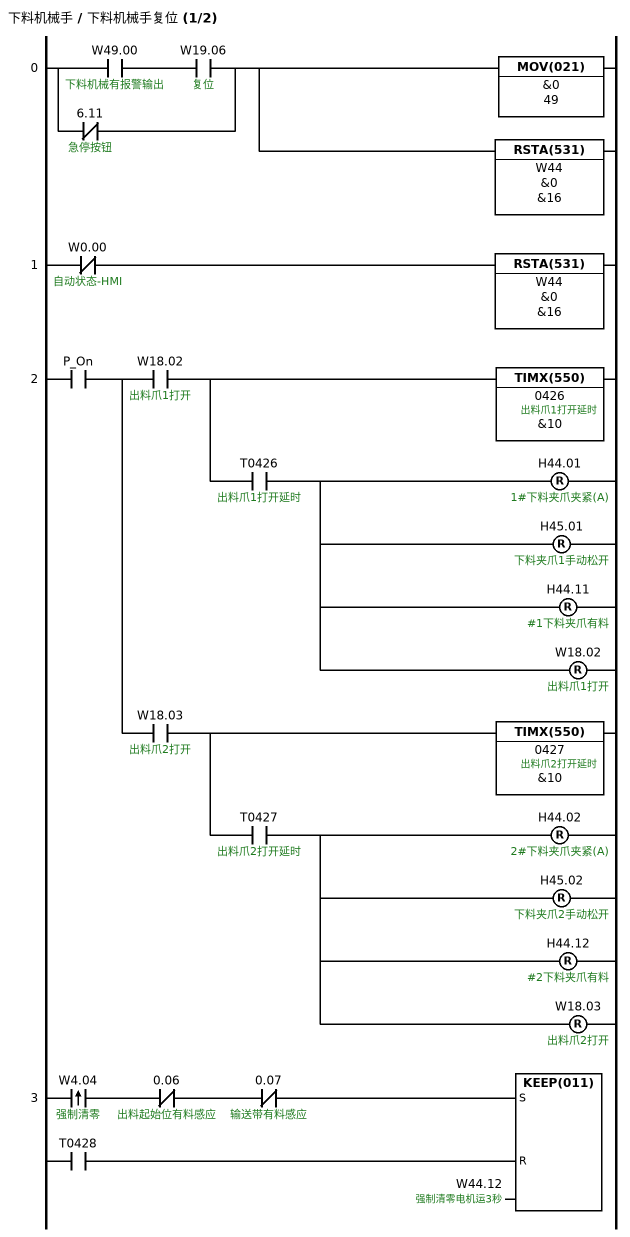
; rung 0
LD W49.00  ; 下料机械有报警输出
AND W19.06  ; 复位
ORNOT 6.11  ; 急停按钮
MOV(021) &0 49
RSTA(531) W44 &0 &16
; rung 1
LDNOT W0.00  ; 自动状态-HMI
RSTA(531) W44 &0 &16
; rung 2
LD P_On
OUT TR0
AND W18.02  ; 出料爪1打开
TIMX(550) 0426 &10  ; 出料爪1打开延时
AND T0426  ; 出料爪1打开延时
RSET H44.01  ; 1#下料夹爪夹紧(A)
RSET H45.01  ; 下料夹爪1手动松开
RSET H44.11  ; #1下料夹爪有料
RSET W18.02  ; 出料爪1打开
LD TR0
AND W18.03  ; 出料爪2打开
TIMX(550) 0427 &10  ; 出料爪2打开延时
AND T0427  ; 出料爪2打开延时
RSET H44.02  ; 2#下料夹爪夹紧(A)
RSET H45.02  ; 下料夹爪2手动松开
RSET H44.12  ; #2下料夹爪有料
RSET W18.03  ; 出料爪2打开
; rung 3
@LD W4.04  ; 强制清零
ANDNOT 0.06  ; 出料起始位有料感应
ANDNOT 0.07  ; 输送带有料感应
LD T0428
KEEP(011) W44.12  ; 强制清零电机运3秒

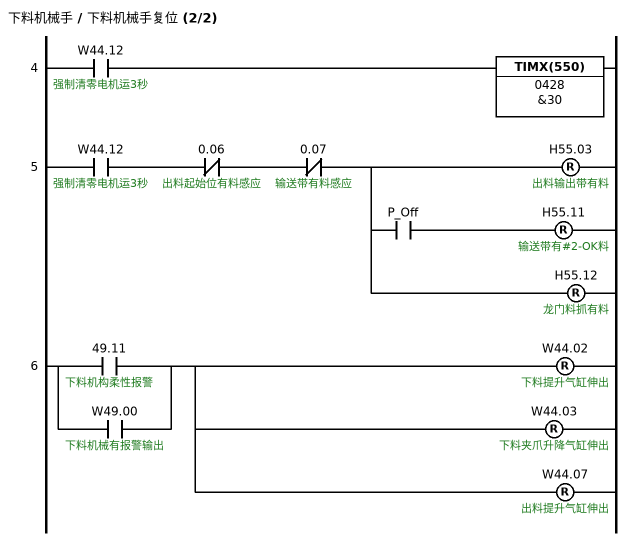
; rung 4
LD W44.12  ; 强制清零电机运3秒
TIMX(550) 0428 &30
; rung 5
LD W44.12  ; 强制清零电机运3秒
ANDNOT 0.06  ; 出料起始位有料感应
ANDNOT 0.07  ; 输送带有料感应
OUT TR0
RSET H55.03  ; 出料输出带有料
AND P_Off
RSET H55.11  ; 输送带有#2-OK料
LD TR0
RSET H55.12  ; 龙门料抓有料
; rung 6
LD 49.11  ; 下料机构柔性报警
OR W49.00  ; 下料机械有报警输出
RSET W44.02  ; 下料提升气缸伸出
RSET W44.03  ; 下料夹爪升降气缸伸出
RSET W44.07  ; 出料提升气缸伸出

### Section END
; rung 0
END(001)

## Program 入盘机械 (cyclic task 5)

### Section 入盘升降_左右轴动作

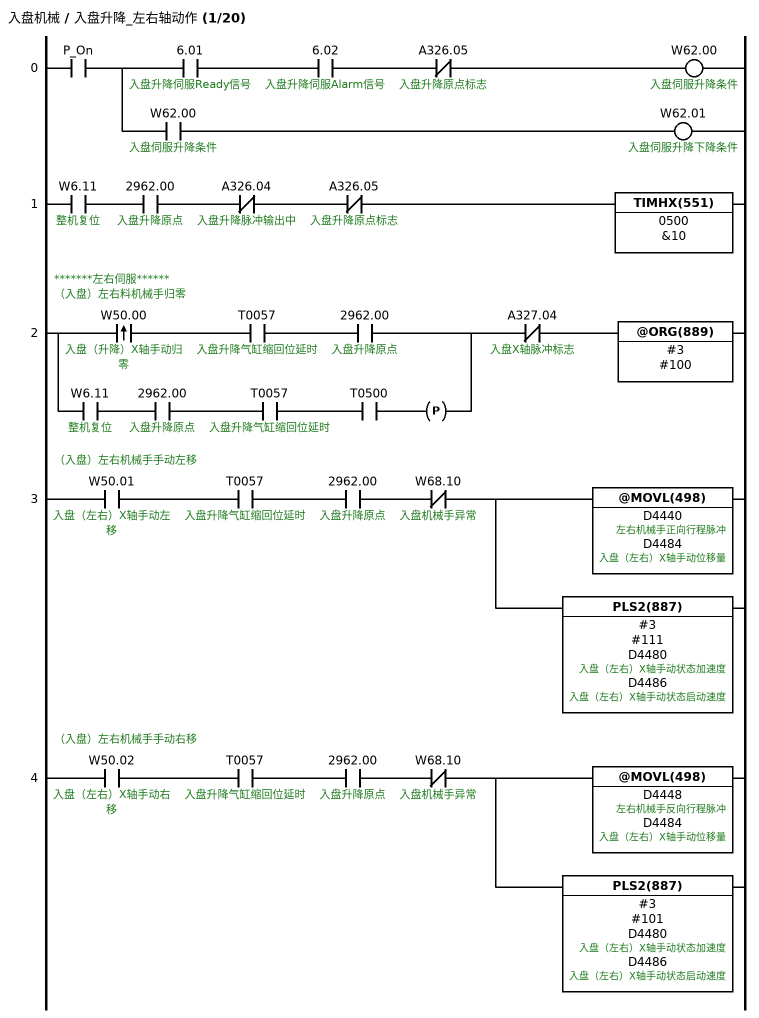
; rung 0
LD P_On
OUT TR0
AND 6.01  ; 入盘升降伺服Ready信号
AND 6.02  ; 入盘升降伺服Alarm信号
ANDNOT A326.05  ; 入盘升降原点标志
OUT W62.00  ; 入盘伺服升降条件
LD TR0
AND W62.00  ; 入盘伺服升降条件
OUT W62.01  ; 入盘伺服升降下降条件
; rung 1
LD W6.11  ; 整机复位
AND 2962.00  ; 入盘升降原点
ANDNOT A326.04  ; 入盘升降脉冲输出中
ANDNOT A326.05  ; 入盘升降原点标志
TIMHX(551) 0500 &10
; rung 2: *******左右伺服****** / （入盘）左右料机械手归零
@LD W50.00  ; 入盘（升降）X轴手动归零
AND T0057  ; 入盘升降气缸缩回位延时
AND 2962.00  ; 入盘升降原点
LD W6.11  ; 整机复位
AND 2962.00  ; 入盘升降原点
AND T0057  ; 入盘升降气缸缩回位延时
AND T0500
UP(521)
ORLD
ANDNOT A327.04  ; 入盘X轴脉冲标志
@ORG(889) #3 #100
; rung 3: （入盘）左右机械手手动左移
LD W50.01  ; 入盘（左右）X轴手动左移
AND T0057  ; 入盘升降气缸缩回位延时
AND 2962.00  ; 入盘升降原点
ANDNOT W68.10  ; 入盘机械手异常
@MOVL(498) D4440 D4484  ; 左右机械手正向行程脉冲, 入盘（左右）X轴手动位移量
PLS2(887) #3 #111 D4480 D4486  ; 入盘（左右）X轴手动状态加速度, 入盘（左右）X轴手动状态启动速度
; rung 4: （入盘）左右机械手手动右移
LD W50.02  ; 入盘（左右）X轴手动右移
AND T0057  ; 入盘升降气缸缩回位延时
AND 2962.00  ; 入盘升降原点
ANDNOT W68.10  ; 入盘机械手异常
@MOVL(498) D4448 D4484  ; 左右机械手反向行程脉冲, 入盘（左右）X轴手动位移量
PLS2(887) #3 #101 D4480 D4486  ; 入盘（左右）X轴手动状态加速度, 入盘（左右）X轴手动状态启动速度

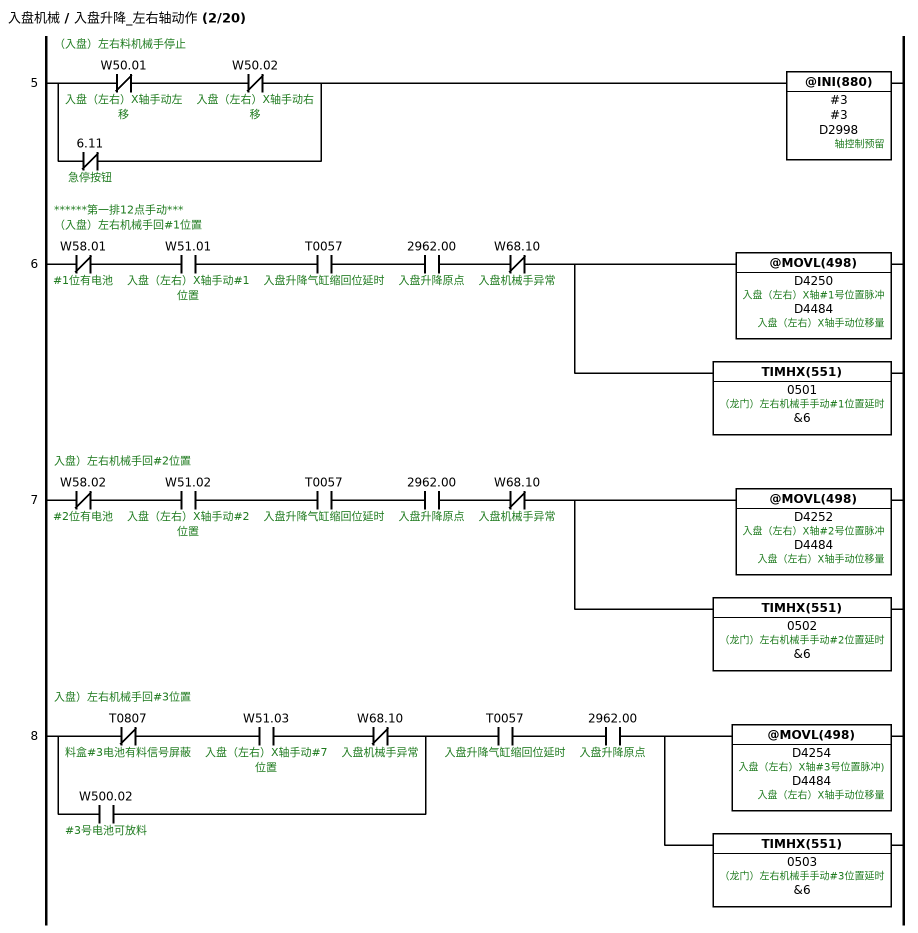
; rung 5: （入盘）左右料机械手停止
LDNOT W50.01  ; 入盘（左右）X轴手动左移
ANDNOT W50.02  ; 入盘（左右）X轴手动右移
ORNOT 6.11  ; 急停按钮
@INI(880) #3 #3 D2998  ; 轴控制预留
; rung 6: ******第一排12点手动*** / （入盘）左右机械手回#1位置
LDNOT W58.01  ; #1位有电池
AND W51.01  ; 入盘（左右）X轴手动#1位置
AND T0057  ; 入盘升降气缸缩回位延时
AND 2962.00  ; 入盘升降原点
ANDNOT W68.10  ; 入盘机械手异常
@MOVL(498) D4250 D4484  ; 入盘（左右）X轴#1号位置脉冲, 入盘（左右）X轴手动位移量
TIMHX(551) 0501 &6  ; （龙门）左右机械手手动#1位置延时
; rung 7: 入盘）左右机械手回#2位置
LDNOT W58.02  ; #2位有电池
AND W51.02  ; 入盘（左右）X轴手动#2位置
AND T0057  ; 入盘升降气缸缩回位延时
AND 2962.00  ; 入盘升降原点
ANDNOT W68.10  ; 入盘机械手异常
@MOVL(498) D4252 D4484  ; 入盘（左右）X轴#2号位置脉冲, 入盘（左右）X轴手动位移量
TIMHX(551) 0502 &6  ; （龙门）左右机械手手动#2位置延时
; rung 8: 入盘）左右机械手回#3位置
LDNOT T0807  ; 料盒#3电池有料信号屏蔽
AND W51.03  ; 入盘（左右）X轴手动#7位置
ANDNOT W68.10  ; 入盘机械手异常
OR W500.02  ; #3号电池可放料
AND T0057  ; 入盘升降气缸缩回位延时
AND 2962.00  ; 入盘升降原点
@MOVL(498) D4254 D4484  ; 入盘（左右）X轴#3号位置脉冲), 入盘（左右）X轴手动位移量
TIMHX(551) 0503 &6  ; （龙门）左右机械手手动#3位置延时

